(* PLC project CoDeSys External Library Template, WAGO e!COCKPIT e!COCKPIT, author 3S - Smart Software Solutions GmbH *)
(* stored: creationDateTime 2019-10-29T12:37:19.7588533, version 3.5.5.30, modificationDateTime 2019-10-29T12:36:39.3744516, organization 3S - Smart Software Solutions GmbH *)
(* Library project template with all possible element types, docu and a sample project structure *)

FUNCTION fnAES256Szyfrowanie : BOOL
  VAR_INPUT
    sKomunikat : alSTRINGKomunikat;
    sKlucz : STRING;
  END_VAR
  VAR_IN_OUT
    intError : INT;
    sKomunikatZaszyfrowany : alSTRINGKomunikat;
  END_VAR

            sKomunikatZaszyfrowany := sKomunikat;
          
END_FUNCTION
